FUNCTION_BLOCK MSb (* Basic FB with empty ECC *)
  (* Standard: 61499-2 *)
  (* Version 1.0, 2025-03-31, 06220625900 *)
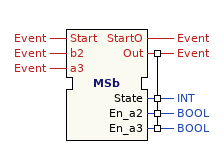
  EVENT_INPUT
    Start;
    b2;
    a3;
  END_EVENT
  EVENT_OUTPUT
    StartO;
    Out WITH State, En_a2, En_a3;
  END_EVENT
  VAR_OUTPUT
    State : INT;
    En_a2 : BOOL;
    En_a3 : BOOL;
  END_VAR
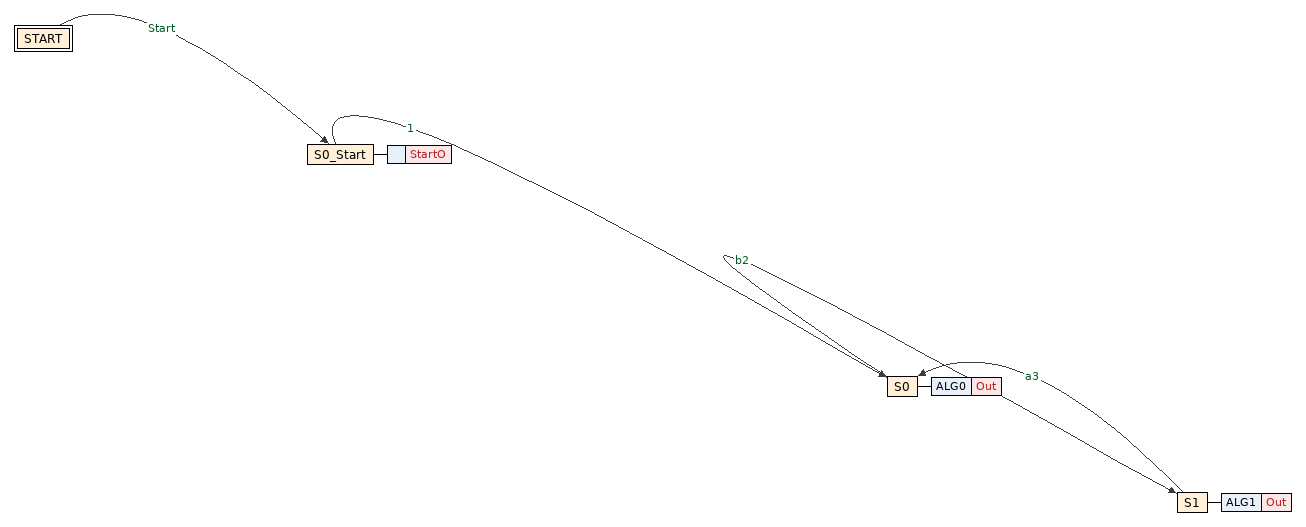
  EC_STATES
    START; (* Initial State *)
    S0_Start : -> StartO;
    S0 : ALG0 -> Out;
    S1 : ALG1 -> Out;
  END_STATES
  EC_TRANSITIONS
    START TO S0_Start := Start;
    S0_Start TO S0 := 1;
    S0 TO S1 := b2;
    S1 TO S0 := a3;
  END_TRANSITIONS
  ALGORITHM ALG0 IN ST:
State:=0;
			En_a2:=TRUE;
			En_a3:=FALSE;
  END_ALGORITHM
  ALGORITHM ALG1 IN ST:
State:=1;
			En_a2:=FALSE;
			En_a3:=TRUE;
  END_ALGORITHM
END_FUNCTION_BLOCK
